FUNCTION_BLOCK FB_InteriorOperationMonitoring
VAR_INPUT
END_VAR
VAR_OUTPUT
END_VAR
VAR
	fb_humiditysensor : FB_HumiditySensor;
	fb_cO2sensor : FB_CO2Sensor;
	fb_temperaturesensor : FB_TemperatureSensor;
	fb_pressuresensor : FB_PressureSensor;
END_VAR

METHOD updateSensorValues
VAR_INPUT
END_VAR
fb_cO2sensor();
fb_humiditysensor();
fb_pressuresensor();
fb_temperaturesensor();

SensorValues.rCO2Value := fb_cO2sensor.getCO2Value;
SensorValues.rHumidity := fb_humiditysensor.getHumidity;
SensorValues.rPressure := fb_pressuresensor.getPressure;
SensorValues.rTemperature := fb_temperaturesensor.getTemperature;
END_METHOD

END_FUNCTION_BLOCK

(* stored: Version 1.1.0.1, ProductVersion 3.1.4024.11
   POU FB_InteriorOperationMonitoring: Id {09ca3a33-707f-4a06-b20c-932141df74ec}, SpecialFunc None
   Method updateSensorValues: Id {0879ac93-2ad3-4ff2-9a0a-e9e0396a0e0b} *)
